PROGRAM database
VAR
END_VAR

END_PROGRAM

(* stored: Version 1.1.0.1, ProductVersion 3.1.4024.12
   POU database: Id {143714b2-f4fe-44a5-9694-f19cd8ef93e2}, SpecialFunc None *)
